FUNCTION_BLOCK FB_MonetTelescopeControl2 EXTENDS FB_AltAzTelescopeControl
VAR_INPUT
	fbFocus				: I_Focus;
	fbCovers			: I_MirrorCovers;
	fbBrake				: I_Brake;	
	fbHydraulics   		: I_Hydraulics;
	fbElevation			: REFERENCE TO FB_ElevationControl;
	fbAzimuth			: REFERENCE TO FB_AzimuthControl;
	fbDerotator			: REFERENCE TO FB_DerotatorControl;
	bEstopTriggered		: BOOL := FALSE;
END_VAR
VAR_OUTPUT
END_VAR
VAR
	bSlewing			: BOOL;
	bStopped			: BOOL;
	bTracking			: BOOL;
	bHomed				: BOOL;
	bReady				: BOOL;
	bBusy				: BOOL;
	tonTrackingDelay	: TON;		// tracking delay
END_VAR

// is telescope slewing?
bSlewing := NOT bTracking AND (fbElevation.fbAxis.InMotion OR fbElevation.fbAxis.InRamp OR
			fbAzimuth.fbAxis.InMotion OR fbAzimuth.fbAxis.InRamp OR
			fbDerotator.fbAxis.InMotion OR fbDerotator.fbAxis.InRamp);
			
// signal must be stable for 5500MS
tonTrackingDelay(
	in := fbElevation.fbAxis.isTracking AND fbAzimuth.fbAxis.isTracking AND fbDerotator.fbAxis.isTracking,
	PT :=T#5500MS, 
	Q => bTracking);
			
// is telescope stopped?
bStopped := (NOT fbElevation.bEnable OR fbElevation.fbAxis.StandStill) AND 
			(NOT fbAzimuth.bEnable OR fbAzimuth.fbAxis.StandStill) AND
			(NOT fbDerotator.bEnable OR fbDerotator.fbAxis.StandStill);
			
// get current coordinates	
fAzimuthCurrent := fbAzimuth.fActualPosition;
fElevationCurrent := fbElevation.fActualPosition;
fDerotatorCurrent := fbDerotator.fActualPosition;

// call super
SUPER^();

// homed, ready, busy
bHomed := fbElevation.bCalibrated AND fbAzimuth.bCalibrated AND fbDerotator.bCalibrated AND fbFocus.Calibrated;
bReady := bHomed AND fbCovers.Opened AND fbElevation.bEnable AND fbAzimuth.bEnable AND fbDerotator.bEnable AND fbBrake.BrakeOpen AND NOT bError;
bBusy  := fbElevation.fbAxis.Busy OR fbAzimuth.fbAxis.Busy OR fbDerotator.fbAxis.Busy OR fbFocus.Busy;

// estop?
IF bEstopTriggered THEN
	fbElevation.Enable := FALSE;
	fbAzimuth.Enable := FALSE;
	fbDerotator.Enable := FALSE;
END_IF

METHOD _Initialize : BOOL
VAR_INPUT
END_VAR
IF NOT bBrakeClearing THEN
	bPowerFailure := TRUE;
	TCSpowerEvent.OnMessage := 'failure: brake clearing not set';
	bPower := FALSE;
ELSIF bError THEN
	bPowerFailure := TRUE;
	TCSpowerEvent.OnMessage := 'Generic error during power on occured.';
	bPower := FALSE;
ELSE
	bPowerFailure := FALSE;		
END_IF

// COVER MUST BE OPENED FOR A SUCCESSFUL WAKE & SHAKE COMMAND!
fbCovers.Open();

// enable elevation, enable azimuth
IF fbCovers.Opened THEN
	fbElevation.Enable := TRUE;
	fbAzimuth.Enable := TRUE;
	fbDerotator.Enable := TRUE;
END_IF

IF fbElevation.Ready AND NOT fbElevation.Calibrated THEN
	fbElevation.HomeAxis := TRUE;
END_IF

IF fbAzimuth.Ready AND NOT fbAzimuth.Calibrated THEN
	fbAzimuth.HomeAxis := TRUE;
END_IF

// enable derotator
IF fbElevation.Ready THEN
	fbDerotator.HomeAxis := fbDerotator.Ready AND NOT fbDerotator.Calibrated;
END_IF

// start calibration of focus after elevation has been calibrated
// this avoids imbalance by the M2 mirror on the elvation during its calibration
IF fbElevation.Calibrated AND NOT fbFocus.Calibrated THEN
	fbFocus.Enable := TRUE;
	fbFocus.HomeAxis := TRUE;
END_IF

IF fbCovers.Opened AND fbElevation.Calibrated AND fbAzimuth.Calibrated AND fbDerotator.Calibrated AND fbFocus.Calibrated THEN
	bPower := FALSE;
	_Initialize := TRUE;
ELSE
	_Initialize := FALSE;
END_IF
END_METHOD

METHOD _Park : BOOL
VAR_INPUT
END_VAR
VAR
	ParkEvent	: FB_Eventlog;
END_VAR
VAR_STAT
	Stage		: USINT := 0;
	LastStage	: USINT := 101;
END_VAR
IF bReset OR bError THEN
	Stage := 0;
END_IF
_Park := FALSE;
CASE Stage OF
	0: 
		fbFocus.Position := telescopeConfig.focusPark;
		IF bError THEN // emergency park
			fbBrake.CloseBrake();
			fbElevation.Enable := FALSE;
			fbAzimuth.Enable := FALSE;
			fbDerotator.Enable := FALSE;	
			fbCovers.Close();	
			Stage := 80;
		END_IF
		Stage := 20;
	20:
		fbElevation.Position := telescopeConfig.elevationPark;
		fbElevation.Velocity := 10.0;
		fbElevation.MoveAxis := TRUE;
		fbAzimuth.Position := telescopeConfig.azimuthPark;
		fbAzimuth.Velocity := 10;
		fbAzimuth.MoveAxis := TRUE;
		fbDerotator.Position := telescopeConfig.derotatorPark;
		fbDerotator.Velocity := 10.0;
		fbDerotator.MoveAxis := TRUE;
		IF fbElevation.Busy AND
			fbAzimuth.Busy AND
			fbDerotator.Busy THEN
				Stage := 40;
		END_IF
	40:
		IF fbElevation.MoveDone THEN
			fbElevation.MoveAxis := FALSE;
		END_IF
		IF fbAzimuth.MoveDone THEN
			fbAzimuth.MoveAxis := FALSE;
		END_IF
		IF fbDerotator.MoveDone THEN
			fbDerotator.MoveAxis := FALSE;
		END_IF
		IF NOT bSlewing THEN // all axis standstill
			Stage := 60;
		END_IF
	60:
		IF NOT fbElevation.Enable AND NOT fbAzimuth.Enable AND NOT fbDerotator.Enable THEN
			stage := 80;
		END_IF

		IF bStopped THEN
			fbElevation.Enable := FALSE;
			fbAzimuth.Enable := FALSE;
			fbDerotator.Enable := FALSE;
		END_IF
		
		fbElevation.bMoveAxis := FALSE;
		fbAzimuth.bMoveAxis := FALSE;
		fbDerotator.bMoveAxis := FALSE;
	80:
		IF fbElevation.Enable OR fbAzimuth.Enable OR fbDerotator.Enable THEN
			stage := 60;
		END_IF
		IF NOT fbBrake.BrakeOpen THEN
			fbCovers.Close();
			fbHydraulics.Enable := FALSE;
		END_IF
		IF fbCovers.Closed THEN
			Stage := 100;
		END_IF
	100:
		_Park := TRUE;
		Stage := 0;	
END_CASE
ParkEvent(Trigger := Stage > LastStage, FormatString := 'Parking progress: %s', OnMessage := USINT_TO_STRING(Stage), comm := comm);
LastStage := Stage;
END_METHOD

METHOD PRIVATE _Slew : BOOL;
VAR_INPUT
END_VAR
VAR
	SlewEvent			:	FB_Eventlog;
	tonCommandTimeout	: TON;
END_VAR
VAR_STAT
	iStage				: USINT;
	iLastStage			: USINT := 101;
END_VAR
_Slew := TRUE;
tonCommandTimeout(IN := iStage < 100, PT := T#600S);
IF tonCommandTimeout.Q THEN
	bError := TRUE;
	//errorid := 16#40;
	//bSlew := FALSE;
	_Slew := FALSE;
	iStage := 0;
END_IF
IF bReset OR bError THEN
	iStage := 0;
END_IF
CASE iStage OF
	0:	
		IF bReady AND bStopped AND NOT bBusy AND NOT bTracking THEN
			iStage := 25;
		END_IF
	25:
		fbElevation.Position := fElevation + PointingModelElevation(fAzimuth, fElevation, EOFF + fElevationOffset, AN_E, AE_E, TF);
		fbElevation.Velocity := 10.0;
		fbElevation.MoveAxis := TRUE;
		fbAzimuth.Position := fAzimuth + PointingModelAzimuth(fAzimuth, fElevation, AOFF + fAzimuthOffset, BNP, AN_A, AE_A, NPAE);
		fbAzimuth.Velocity := 10.0;
		fbAzimuth.MoveAxis := TRUE;
		fbDerotator.Position := fElevation + fDerotatorOffset;
		fbDerotator.Velocity := 10.0;
		fbDerotator.MoveAxis := TRUE;
		IF fbElevation.Busy AND fbAzimuth.Busy AND fbDerotator.Busy THEN
			iStage := 50;
		END_IF
	50:
		IF fbElevation.MoveDone THEN
			fbElevation.bMoveAxis := FALSE;
		END_IF
		
		IF fbAzimuth.MoveDone THEN
			fbAzimuth.MoveAxis := FALSE;
		END_IF

		IF fbDerotator.MoveDone THEN
			fbDerotator.MoveAxis := FALSE;
		END_IF
		IF NOT bSlewing AND bStopped THEN // all axis standstill
			iStage := 100;
		END_IF
	100:
		fbElevation.MoveAxis := FALSE;
		fbAzimuth.MoveAxis := FALSE;
		fbDerotator.MoveAxis := FALSE;
		fRightAscension := fRightAscensionCalc;
		fDeclination := fDeclinationCalc;
		_Slew := FALSE;
END_CASE

SlewEvent(Trigger := iStage > iLastStage, FormatString := 'Slew progress: %s', OnMessage := USINT_TO_STRING(iStage), comm := comm);
iLastStage := iStage;
END_METHOD

METHOD _Stop : BOOL
VAR_INPUT
END_VAR
fbElevation.StopAxis := TRUE;
fbAzimuth.StopAxis := TRUE;
fbDerotator.StopAxis := TRUE;
_Stop := FALSE;

IF bStopped THEN
	fbElevation.StopAxis := FALSE;
	fbAzimuth.StopAxis := FALSE;
	fbDerotator.StopAxis := FALSE;
	_Stop := TRUE;
END_IF
END_METHOD

END_FUNCTION_BLOCK

(* stored: Version 1.1.0.1, ProductVersion 3.1.4024.15
   POU FB_MonetTelescopeControl2: Id {392c90d3-a441-4c8d-a752-42b25b49f5cd}, SpecialFunc None
   Method _Initialize: Id {b82ca6ca-e327-451f-ab83-9e7ad8e568da}
   Method _Park: Id {b753730c-f439-4fd9-a185-d431d3c6a732}
   Method _Slew: Id {b97e5388-b217-43fc-a742-07bcca507bbe}
   Method _Stop: Id {25d1a575-544b-48f0-8dce-8d30aad96001} *)
